Staubli VAL3: IsSetValue.pgx

public program IsSetValue()
begin
  //  x_bOk=true
  //  if save:nBoxType==1
  //
  //    if  sml:box[x_sName].nKeySafeNum[0]==0
  //
  //
  //    endIf
  //  elseIf save:nBoxType==2
  //
  //  endIf
end
